FUNCTION_BLOCK FB_ExtruderRef
VAR_INPUT
END_VAR
VAR
	rFactorDistance		: REAL;
	rFactorFeed			: REAL;
	nFeedOrgin			: DINT;	//µm/s
	nCompFeedOrgin		: DINT;	//µm/s
	nRelaxFeedOrgin		: DINT;	//µm/s
	nDistanceOrgin		: DINT;	//µm
	nCompDistanceOrgin	: DINT;	//µm
	nRelaxDistanceOrgin	: DINT;	//µm
	
	//Umgerechnete Werte
	nFeedCalc			: DINT; // 1/100tel RPM
	nCompFeedCalc		: DINT; // 1/100tel RPM
	nRelaxFeedCalc		: DINT; // 1/100tel RPM
	nDistanceCalc		: DINT;	// µm
	nCompDistanceCalc	: DINT;	// µm
	nRelaxDistanceCalc	: DINT;	// µm	
END_VAR
VAR_OUTPUT
END_VAR

//Basisklasse

PROPERTY P_bError : BOOL
GET
END_GET
END_PROPERTY

PROPERTY P_bIsActive : BOOL
GET
END_GET
END_PROPERTY

PROPERTY P_bIsLocked : BOOL
GET
END_GET
END_PROPERTY

PROPERTY P_nCompDistanceCalc : DINT
GET
P_nCompDistanceCalc := nCompDistanceCalc;
END_GET
END_PROPERTY

PROPERTY P_nCompDistanceOrgin : DINT
GET
P_nCompDistanceOrgin := nCompDistanceOrgin;
END_GET
SET
nCompDistanceOrgin := P_nCompDistanceOrgin;
nCompDistanceCalc := REAL_TO_DINT(rFactorDistance * DINT_TO_REAL(nCompDistanceOrgin));
END_SET
END_PROPERTY

PROPERTY P_nCompFeedCalc : DINT
GET
P_nCompFeedCalc := nCompFeedCalc;
END_GET
END_PROPERTY

PROPERTY P_nCompFeedOrgin : DINT
GET
P_nCompFeedOrgin := nCompFeedOrgin;
END_GET
SET
nCompFeedOrgin := P_nCompFeedOrgin;
nCompFeedCalc := REAL_TO_DINT(rFactorFeed * DINT_TO_REAL(nCompFeedOrgin));
END_SET
END_PROPERTY

PROPERTY P_nCurrentPos : DINT
GET
END_GET
END_PROPERTY

PROPERTY P_nDistanceCalc : DINT
GET
P_nDistanceCalc := nDistanceCalc;
END_GET
END_PROPERTY

PROPERTY P_nDistanceOrgin : DINT
GET
P_nDistanceOrgin := nDistanceOrgin;
END_GET
SET
nDistanceOrgin := P_nDistanceOrgin;
nDistanceCalc := REAL_TO_DINT(rFactorDistance * DINT_TO_REAL(nDistanceOrgin));
END_SET
END_PROPERTY

PROPERTY P_nFeedCalc : DINT
GET
P_nFeedCalc := nFeedCalc;
END_GET
END_PROPERTY

PROPERTY P_nFeedOrgin : DINT
GET
P_nFeedOrgin := nFeedOrgin;
END_GET
SET
nFeedOrgin := P_nFeedOrgin;
nFeedCalc := REAL_TO_DINT(rFactorFeed * DINT_TO_REAL(nFeedOrgin));
END_SET
END_PROPERTY

PROPERTY P_nRelaxDistanceCalc : DINT
GET
P_nRelaxDistanceCalc := nRelaxDistanceCalc;
END_GET
END_PROPERTY

PROPERTY P_nRelaxDistanceOrgin : DINT
GET
P_nRelaxDistanceOrgin := nRelaxDistanceOrgin;
END_GET
SET
nRelaxDistanceOrgin := P_nRelaxDistanceOrgin;
nRelaxDistanceCalc := REAL_TO_DINT(rFactorDistance * DINT_TO_REAL(nRelaxDistanceOrgin));
END_SET
END_PROPERTY

PROPERTY P_nRelaxFeedCalc : DINT
GET
P_nRelaxFeedCalc := nRelaxFeedCalc;
END_GET
END_PROPERTY

PROPERTY P_nRelaxFeedOrgin : DINT
GET
P_nRelaxFeedOrgin := nRelaxFeedOrgin;
END_GET
SET
nRelaxFeedOrgin := P_nRelaxFeedOrgin;
nRelaxFeedCalc := REAL_TO_DINT(rFactorFeed * DINT_TO_REAL(nRelaxFeedOrgin));
END_SET
END_PROPERTY

PROPERTY P_rFactorDistance : REAL
GET
P_rFactorDistance := rFactorDistance;
END_GET
SET
rFactorDistance := P_rFactorDistance;
END_SET
END_PROPERTY

PROPERTY P_rFactorFeed : REAL
GET
P_rFactorFeed := rFactorFeed;
END_GET
SET
rFactorFeed := P_rFactorFeed;
END_SET
END_PROPERTY

END_FUNCTION_BLOCK

(* stored: Version 1.1.0.1, ProductVersion 3.1.4022.7
   POU FB_ExtruderRef: Id {cc13f0ed-bb1c-4ba8-8fc3-fb04af90d564}, SpecialFunc None
   Property P_bError: Id {a90aa48c-3e84-437b-b36b-7701c9a26430}
   Get Get: Id {6b65e6a9-f3cc-4540-81a4-f48fa7f7be46}
   Property P_bIsActive: Id {a2846892-759b-4962-9d83-764df0747dd6}
   Get Get: Id {3edad862-2463-477f-a7f4-58a1bdd8625f}
   Property P_bIsLocked: Id {136d906a-8ef0-42fa-85df-aebfb25873cd}
   Get Get: Id {c05d1e06-e56c-4ad4-850d-67d234557d86}
   Property P_nCompDistanceCalc: Id {d7932961-be6a-4a56-a696-9365c1284f6f}
   Get Get: Id {9ada38a7-0350-48ce-b2d1-9b66c48d104d}
   Property P_nCompDistanceOrgin: Id {5e1885b2-a4dc-41fc-977c-d2e9e0e4fdaf}
   Get Get: Id {8f618551-faf6-42e6-ba50-21c91f759d18}
   Set Set: Id {755d6107-2010-4731-afb6-9bb98806dc56}
   Property P_nCompFeedCalc: Id {1be23e13-c82a-4621-8a81-b8009d3c22ef}
   Get Get: Id {3983d0d5-4248-46a2-8411-b3868de2851b}
   Property P_nCompFeedOrgin: Id {b6b47049-4937-4eb2-833a-43a852e0d1f7}
   Get Get: Id {8091d12e-8113-45a6-b1d9-10015d40649c}
   Set Set: Id {95087693-fe72-4de1-bfee-5a26515dd631}
   Property P_nCurrentPos: Id {0269be9b-31e5-4849-b342-648d45226c4a}
   Get Get: Id {26c5381f-1be5-45cf-a72b-f30119f83a3d}
   Property P_nDistanceCalc: Id {194f4c34-07e2-41c6-b67c-6d05c2397e15}
   Get Get: Id {46b74109-a82d-45e6-a491-cfe87a367f3e}
   Property P_nDistanceOrgin: Id {095df1c9-fa12-481a-9952-6e3ac88cdbba}
   Get Get: Id {e590f7e7-20e9-40ea-9cc4-7750b0cc1a97}
   Set Set: Id {412be54d-7c51-43da-a802-726b757f3afd}
   Property P_nFeedCalc: Id {60155019-64d8-4050-b091-340b26cd2149}
   Get Get: Id {008b4e81-504b-48ed-8021-d8865e125793}
   Property P_nFeedOrgin: Id {2c9c9e45-b81f-452f-8dc1-41a87f235b1d}
   Get Get: Id {6f8027b2-d396-4791-bdf7-f0a96025ced3}
   Set Set: Id {d7755730-32f8-4860-b672-2472c2a601ae}
   Property P_nRelaxDistanceCalc: Id {b331b8d2-581b-4a10-a2a1-059efc592042}
   Get Get: Id {4de7f85f-8a97-44cc-8510-25ea919cbb07}
   Property P_nRelaxDistanceOrgin: Id {589dcb0d-27a6-4ad4-bb9e-919c15461576}
   Get Get: Id {a9b6788d-fb2a-4218-975c-f6ba3e606045}
   Set Set: Id {0799025d-c435-4bc8-a22a-eacb42bc2aa7}
   Property P_nRelaxFeedCalc: Id {04d8e9d7-c3de-4fb3-ac71-4d617f15ade4}
   Get Get: Id {974c1f3c-3ed9-4f74-b66a-4443b3b8b76b}
   Property P_nRelaxFeedOrgin: Id {1ebfa167-d1b2-4c39-a5fb-74cc5d6bfc95}
   Get Get: Id {23ec6873-736e-4c58-9455-222b20bba739}
   Set Set: Id {fe95ab7c-79b2-41dc-8ebb-ff37cdcd639a}
   Property P_rFactorDistance: Id {20def287-7612-4379-8c6a-5a20ad96f60b}
   Get Get: Id {5cab9da3-fe0b-46c5-95ef-912d946152b5}
   Set Set: Id {9e020033-dd7a-43da-ace3-c8d7a0c600ab}
   Property P_rFactorFeed: Id {6825f398-a927-4562-b2d1-db6542088ae8}
   Get Get: Id {909411c2-61d4-4d6c-976e-202186ccfe42}
   Set Set: Id {db2acedd-8ed4-47a6-8b23-030287511c0a} *)
